// TIA Portal V17 export
// export: Created 2024-09-15T12:29:55.1114546Z, ExportSetting WithDefaults, DisplayName Totally Integrated Automation Portal, DisplayVersion V17, DisplayName TIA Portal Openness, DisplayVersion V17, DisplayName TIA Portal Version Control Interface, DisplayVersion V17, DisplayName STEP 7 Professional, DisplayVersion V17, DisplayName STEP 7 Safety, DisplayVersion V17, DisplayName WinCC Professional, DisplayVersion V17
DATA_BLOCK "PRG_Order_DB"   // DB25
AUTHOR : A.Schaefer
VERSION : 0.1
// stored: AutoNumber true, DBAccessibleFromOPCUA true, DBAccessibleFromWebserver true, InstanceOfName PRG_Order, InstanceOfType FB
"PRG_Order"
   // VAR
   //    lx_Init { ExternalAccessible := 'False'; ExternalVisible := 'False'; ExternalWritable := 'False'} : Bool;
   //    li_StepCase { ExternalAccessible := 'False'; ExternalVisible := 'False'; ExternalWritable := 'False'} : Int;
   //    lldt_ts_old { ExternalAccessible := 'False'; ExternalVisible := 'False'; ExternalWritable := 'False'} : LDT;
   //    ldt_MQTT { ExternalAccessible := 'False'; ExternalVisible := 'False'; ExternalWritable := 'False'} : Date_And_Time;
   //    li_Return_LDT { ExternalAccessible := 'False'; ExternalVisible := 'False'; ExternalWritable := 'False'} : Int;
   //    lfb_TON_Wait { ExternalAccessible := 'False'; ExternalVisible := 'False'; ExternalWritable := 'False'} : TON_TIME;
   //    lx_Start_TON_Wait { ExternalAccessible := 'False'; ExternalVisible := 'False'; ExternalWritable := 'False'} : Bool;
   // END_VAR
BEGIN
END_DATA_BLOCK
